// TIA Portal V19 export
TYPE "LAF_typePlasticWorkstationEm5ProcessValuesHmi"
// stored: Access Published
   STRUCT
      pieceCount : DInt;
   END_STRUCT;
END_TYPE
